// TIA Portal V18 export
VAR_GLOBAL   // PLC tag table "00 Costanti MASTER"
END_VAR
VAR_GLOBAL CONSTANT   // user constants
   N_ZONE : DInt := 5;   // Numero di zone massime presenti nelle linee
   N_DS : DInt := 50;   // Numero di dati per sezione
   N_SAFETYDEVICE : DInt := 15;   // Numero di dispositivi di sicurezza per sezione
   N_STAZIONI : DInt := 20;   // Numero max stazioni linea
   N_MaxAttuatoriStz : Int := 10;   // numero massimo attuatori per stazione
   N_MaxMonitoraggi : Int := 30;
   N_MaxMonitoraggiPag : Int := 5;
   N_HMI : DInt := 7;   // Numero pannelli HMI da 0 a 5
   N_AssiAAA : Int := 10;
   N_PrgValvole : Int := 5;   // Numero programmi valvole proporzionali
END_VAR
